Staubli VAL3: Instruction.pjx

--- Instruction.pjx ---
Parameters version=s7.2.1 stackSize=5000 millimeterUnit=true
Data file=Instruction.dtx

--- Instruction.dtx ---
public bool bIsTraj
public string sPath
public string sID
public bool bUseOnPoint
public num nIndex
